// TwinCAT 3 PLC project Untitled1
// ProgramVersion: 3.1.4024.0
// libraries:
//   Tc2_Standard, * (Beckhoff Automation GmbH)
//   Tc2_System, * (Beckhoff Automation GmbH)
//   Tc3_Module, * (Beckhoff Automation GmbH)
// project tree:
//   GVLs/POUs/ MAIN.TcPOU
//   / PlcTask.TcTTO

CONFIGURATION Untitled1
    RESOURCE PLC ON TwinCAT3
        TASK PlcTask(INTERVAL := T#10ms, PRIORITY := 20);
        PROGRAM MAIN WITH PlcTask : MAIN;
    END_RESOURCE
END_CONFIGURATION

// ---- GVLs/POUs/MAIN.TcPOU
PROGRAM MAIN
VAR
	//vnt 1
	bTest_1: BOOL;
	//CNT 2
	bTest_2: BOOL;
END_VAR

END_PROGRAM
